// Brief: Mounting Instrument
FUNCTION_BLOCK PUBLIC FB_SlaveCtrlMountInstru EXTENDS FB_SlaveArmCtrlBase
VAR
	// mount status
	m_instruMountStatus :INT := 0;
	m_scopeMountStatus :INT := 0;
	m_ultrasoundMountStatus :INT :=0 ;
	
	// flag if joint is mounted
	m_jointMounted :ARRAY[1..5] OF BOOL := [5(FALSE)];
	
	// instrument mount motion range
	m_mountMotionAng :Vec5d :=[5(pi)];
	
	// instrument mount direction
	m_mountDir :Vec5i :=[1, 1, 1, 1, 1];
	
	// mount motion planning
	m_jntOTG :ARRAY[1..5] OF FB_secOrdTrajFilter;
	m_instruMountVel :LREAL := 4*PI;
	m_instruMountAcc :LREAL := 8*PI;
	
	//Joint 4 half-range angle of instrument
	m_instruJnt4HalfRangeAng :LREAL := 323*g_deg2Rad;
	
	// joint current threshold which indicate panel is buckled with instrument
	m_maxJntCurrent :Vec5d := [150, 150, 150, 180, 180];
	
	// command mount motion
	m_targetMountPos :Vec8d;
	
	// instrument zero position
	m_instruZeroDeviation :Vec5d;
	
	//ultrasound knife Reduce the current rotation Angle  J3
	m_ultraKnifeRotaAngleJ3 :LREAL := 30*g_deg2Rad;
	
	// ultrasound knife rotate angle zero position
	m_ultraKnifeRotAngZeroPos :LREAL := 4.50567;
	
	// joint position error
	m_jntPosErr :Vec5d;
	
	// endoscope motion angle to original position
	m_scopeJnt4CenterMotionAng :LREAL :=175*g_deg2Rad;
	m_scopeJnt5CenterMotionAng :LREAL :=150*g_deg2Rad;
	
	//instrument clamp error Id
	m_instruClampErrId : UINT;
	m_instruClampTime : LREAL;
	m_noCurrentTime : LREAL :=3;
	m_notReturnToZero : LREAL :=5;
END_VAR

// override this function in each exact controller
METHOD PROTECTED calcCmdJntPos : BOOL
VAR_IN_OUT CONSTANT
	i_endoscopePose : ST_Frame;
	i_masterStatus :ST_MasterStatus;
	i_setupStatus: ST_SetupStatus;
	i_slaveArm :FB_SlaveArm;
END_VAR

VAR 
END_VAR
// return directly if instrument/endoscope is not readed
IF i_slaveArm.instrument.onChipData.m_Error OR m_instruClampErrId >0  THEN
	return;
END_IF

IF i_slaveArm.instrument.onChipData.m_InstruReadSucceed AND InstruType_endoscope = i_slaveArm.instrument.m_instruType THEN
	mountEndoscope(i_slaveArm);
ELSIF i_slaveArm.instrument.onChipData.m_InstruReadSucceed AND (InstruType_UltrasoundKnifeS = i_slaveArm.instrument.m_instruType OR InstruType_UltrasoundKnifeU = i_slaveArm.instrument.m_instruType) THEN
	mountUltraKnife(i_slaveArm);
ELSE
	mountInstrument(i_slaveArm);
END_IF
m_instruClampErrId := instruClampStatus(i_slaveArm);
END_METHOD

METHOD PUBLIC init : BOOL
VAR_IN_OUT CONSTANT
	i_slaveArm	:FB_SlaveArm;
END_VAR
VAR_IN_OUT 
	r_slaveArmCtrlCmd :ST_SlaveArmCtrlCmds;
END_VAR

VAR
	i : INT;
END_VAR
// check if to hold the command joint position unchanged
m_holdLastCmds := checkToHoldLastCmds(i_slaveArm);

SUPER^.Init(i_slaveArm,r_slaveArmCtrlCmd);
m_jntOPMode[4] := DriverOPMode_PosTrq;
m_jntOPMode[5] := DriverOPMode_PosTrq;
m_jntOPMode[6] := DriverOPMode_PosTrq;
m_jntOPMode[7] := DriverOPMode_PosTrq;
m_jntOPMode[8] := DriverOPMode_PosTrq;

FOR i:=1 TO 5 DO
	m_targetMountPos[i+3]:=m_cmdJntPos[i+3];
	m_jntOTG[i].init(m_targetMountPos[i+3], 0,m_instruMountVel, m_instruMountAcc, g_slaveArmCtrlCycleTime);
	m_jointMounted[i]:=FALSE;
END_FOR

m_instruMountStatus:=0;
m_scopeMountStatus:=0;
m_ultrasoundMountStatus:=0;
m_instruClampErrId := 0;
m_instruClampTime := 0;
// update commands to arm
copyCmds(r_slaveArmCtrlCmd);
END_METHOD

PROPERTY instruClampErrId :  UINT
GET
instruClampErrId := m_instruClampErrId;
END_GET
END_PROPERTY

METHOD instruClampStatus : UINT
VAR_IN_OUT CONSTANT
	i_slaveArm :FB_SlaveArm;
END_VAR
//m_instruClampErrId=1 instrumen clamp the current does not reach the set value
//m_instruClampErrId=2 instrumen clamp position does not return to zero
m_instruClampTime := LIMIT(0,m_instruClampTime + g_slaveArmCtrlCycleTime,10);
IF i_slaveArm.instrument.onChipData.m_InstruReadSucceed THEN
	IF InstruType_endoscope = i_slaveArm.instrument.m_instruType THEN
		IF (m_scopeMountStatus=0 OR m_scopeMountStatus=1) AND m_instruClampTime>=m_noCurrentTime  THEN
			instruClampStatus := 1;
		ELSIF m_scopeMountStatus=3 AND m_instruClampTime>=m_notReturnToZero  THEN
			instruClampStatus := 2;
		END_IF
		
	ELSIF (InstruType_UltrasoundKnifeS = i_slaveArm.instrument.m_instruType OR InstruType_UltrasoundKnifeU = i_slaveArm.instrument.m_instruType) THEN
		IF (m_ultrasoundMountStatus=0) AND m_instruClampTime>=m_noCurrentTime  THEN
			instruClampStatus := 1;
		ELSIF (m_scopeMountStatus=3) AND m_instruClampTime>=m_notReturnToZero  THEN
			instruClampStatus := 2;
		END_IF
			
	ELSE
		IF (m_instruMountStatus=0) AND m_instruClampTime>=m_noCurrentTime  THEN
			instruClampStatus := 1;
		ELSIF (m_instruMountStatus=3) AND m_instruClampTime>=m_notReturnToZero  THEN
			instruClampStatus := 2;
		END_IF
	END_IF
END_IF
END_METHOD

METHOD mountEndoscope : BOOL
VAR_IN_OUT CONSTANT
	i_slaveArm :FB_SlaveArm;
END_VAR

VAR 
	i :INT;
	curJntPos :Vec8d;
END_VAR
curJntPos := i_slaveArm.curJntPos;

CASE m_scopeMountStatus OF
	//fix scope lock joint(joint 7)
	0:
		// other joints stay still
		FOR i:=1 TO 3 DO
			m_jointMounted[i] := TRUE;
			m_targetMountPos[i+3]:=curJntPos[i+3];
			m_jntOTG[i].init(m_targetMountPos[i+3], 0,m_instruMountVel, m_instruMountAcc, g_slaveArmCtrlCycleTime);
		END_FOR
	
		// check if buckled
		m_jointMounted[4]:=FALSE; 
		m_jointMounted[5]:=FALSE; 
		IF ABS(i_slaveArm.filtJntCurrent[7])> m_maxJntCurrent[4] THEN 
			m_jointMounted[4]:=TRUE;
			m_targetMountPos[7]:=curJntPos[7];
			m_jntOTG[4].init(m_targetMountPos[7], 0,m_instruMountVel, m_instruMountAcc, g_slaveArmCtrlCycleTime);
			m_scopeMountStatus:=1;
		ELSE
			m_targetMountPos[7]:=curJntPos[7]+m_mountMotionAng[4];
		END_IF

	1: // buckle scope rotate joint (joint 8)
		m_jointMounted[5]:=FALSE; 
		IF ABS(i_slaveArm.filtJntCurrent[8])> m_maxJntCurrent[5] THEN 
			m_jointMounted[5]:=TRUE;
			m_targetMountPos[8]:=curJntPos[8];
			m_jntOTG[5].init(m_targetMountPos[8], 0,m_instruMountVel, m_instruMountAcc, g_slaveArmCtrlCycleTime);
			m_scopeMountStatus:=2;
		ELSE
			m_targetMountPos[8]:=curJntPos[8]+m_mountMotionAng[5];
		END_IF
	

	2:// move back to zero position
		m_targetMountPos[7]:= curJntPos[7]-m_scopeJnt4CenterMotionAng;
		m_targetMountPos[8]:= curJntPos[8]-m_scopeJnt5CenterMotionAng;
		m_scopeMountStatus :=3;
		
		
	3:
		IF ABS(m_targetMountPos[7]-curJntPos[7]) <GVL_SlaveControlParameters.g_jntCtrlAngTolHigh AND 
				ABS(m_targetMountPos[8]-curJntPos[8]) <GVL_SlaveControlParameters.g_jntCtrlAngTolHigh THEN
			// record current joint position as offset for instrument
			i_slaveArm.instrument.initInstruJntPos(i_slaveArm.curJntPos);
			m_isFinished := TRUE;
		END_IF
		
END_CASE

// traj plan
FOR i:=1 TO 5 DO
	m_jntOTG[i].run(m_targetMountPos[i+3],0.0, o_cmdAcc=>m_cmdJntAcc[3+i],o_cmdVel=>m_cmdJntVel[3+i],o_cmdPos=>m_cmdJntPos[i+3]);
END_FOR
END_METHOD

METHOD mountInstrument : BOOL
VAR_IN_OUT CONSTANT
	i_slaveArm :FB_SlaveArm;
END_VAR

VAR 
	i :INT;
	curJntPos :Vec8d;
END_VAR
curJntPos := i_slaveArm.curJntPos;

// joint4 stay still if instrument has only on finger
IF i_slaveArm.instrument.m_isSingleFinger THEN
	m_jointMounted[1]:=TRUE;
END_IF

CASE m_instruMountStatus OF
	// To lock panel with instrument
	0:
		//buckle panel with instrument
		FOR i:=1 TO 4 DO
			// check if buckled 
			IF ABS(i_slaveArm.filtJntCurrent[i+3])> m_maxJntCurrent[i] THEN 
				m_jointMounted[i]:=TRUE;
				m_targetMountPos[i+3]:=curJntPos[i+3];
				m_jntOTG[i].init(m_targetMountPos[i+3], 0,m_instruMountVel, m_instruMountAcc, g_slaveArmCtrlCycleTime);
			END_IF
			
			// set target joint position
			IF FALSE = m_jointMounted[i] THEN
				IF i = 4 THEN
					m_targetMountPos[i+3]:=curJntPos[i+3]+m_mountMotionAng[i];
				ELSE
					m_targetMountPos[i+3]:=curJntPos[i+3]-m_mountMotionAng[i];
				END_IF
				
			END_IF
		END_FOR
		
		
		// check transition condition
		IF (m_jointMounted[1] AND m_jointMounted[2] AND m_jointMounted[3] AND m_jointMounted[4])  THEN
			IF i_slaveArm.instrument.onChipData.m_InstruReadSucceed THEN//Check whether the data is read successfully
				m_instruMountStatus:=1;
			END_IF
		END_IF
	
	1:// calculation deviates from the instrument zero position
		FOR i:=1 TO 4 DO
			m_instruZeroDeviation[i] :=  i_slaveArm.linkSingle[i+3] - i_slaveArm.instrument.onChipData.m_InstruPos[i];
		END_FOR
		m_instruMountStatus :=2;
	
	
	2:// move back to zero position
		FOR i:=1 TO 3 DO//J1-3
			IF m_instruZeroDeviation[i]>pi THEN
				m_instruZeroDeviation[i] := m_instruZeroDeviation[i] - 2*PI;
			ELSIF m_instruZeroDeviation[i]<-pi THEN
				m_instruZeroDeviation[i] := m_instruZeroDeviation[i] + 2*PI;
			END_IF
		END_FOR
		
		//joint4
		IF m_instruZeroDeviation[4]>0 AND m_instruZeroDeviation[4] < pi THEN
			m_instruZeroDeviation[4] := m_instruZeroDeviation[4] - 2*pi;
		ELSIF m_instruZeroDeviation[4]<0 AND m_instruZeroDeviation[4] > -pi THEN
			m_instruZeroDeviation[4] := m_instruZeroDeviation[4] + 2*pi;
		END_IF
		
		// set target joint position
		FOR i:=1 TO 4 DO
			m_targetMountPos[i+3]:=curJntPos[i+3] - m_instruZeroDeviation[i];
		END_FOR
		m_instruMountStatus :=3;
	
	3: // make fingers is closed
		//m_instruMountStatus :=4;
		FOR i:=1 TO 4 DO 
			m_jointMounted[i]:=FALSE;
			m_jntPosErr[i]:=m_targetMountPos[i+3]-curJntPos[i+3];
			IF ABS(m_jntPosErr[i]) <GVL_SlaveControlParameters.g_jntCtrlAngTolLow OR 
					ABS( i_slaveArm.linkSingle[i+3] - i_slaveArm.instrument.onChipData.m_InstruPos[i]) <5*g_deg2rad THEN
				m_jointMounted[i]:=TRUE;
				//EXIT;
			END_IF
		END_FOR
		
		IF ABS(i_slaveArm.filtJntCurrent[7])> m_maxJntCurrent[4] AND ABS(i_slaveArm.curJntVel[7])< 1*g_deg2rad AND
				ABS( i_slaveArm.linkSingle[7] - i_slaveArm.instrument.onChipData.m_InstruPos[4]) >10*g_deg2rad AND NOT m_jointMounted[4] THEN 
			m_instruZeroDeviation[4] :=  i_slaveArm.linkSingle[7] - i_slaveArm.instrument.onChipData.m_InstruPos[4];
			m_jointMounted[4]:=TRUE;
			IF m_instruZeroDeviation[4]>=0 AND m_instruZeroDeviation[4] < pi THEN
				m_instruZeroDeviation[4] := m_instruZeroDeviation[4] - 2*pi;
			ELSIF m_instruZeroDeviation[4]<0 AND m_instruZeroDeviation[4] > -pi THEN
				m_instruZeroDeviation[4] := m_instruZeroDeviation[4] + 2*pi;	
			END_IF
		ELSE
			m_instruZeroDeviation[4] := 0;
		END_IF
		
		IF (m_jointMounted[1] AND m_jointMounted[2] AND m_jointMounted[3] AND m_jointMounted[4])  THEN
			m_instruMountStatus :=4;
		END_IF
		
		IF m_instruMountStatus =4 AND NOT( i_slaveArm.instrument.m_isSingleFinger) THEN
			m_targetMountPos[4] := curJntPos[4]+g_gripperCloseAng;
			m_targetMountPos[5] := curJntPos[5]+g_gripperCloseAng;
			m_targetMountPos[7] := curJntPos[7]-m_instruZeroDeviation[4];
		END_IF
		
	4:
		m_isFinished :=  ABS(m_targetMountPos[4]-curJntPos[4]) < GVL_SlaveControlParameters.g_jntCtrlAngTolLow AND
			 ABS(m_targetMountPos[5]-curJntPos[5]) < GVL_SlaveControlParameters.g_jntCtrlAngTolLow AND ABS(m_targetMountPos[7]-curJntPos[7]) < GVL_SlaveControlParameters.g_jntCtrlAngTolLow;
			 
		// record current joint position as offset for instrument
		i_slaveArm.instrument.initInstruJntPos(i_slaveArm.curJntPos);

END_CASE

// traj plan
FOR i:=1 TO 4 DO
	m_jntOTG[i].run(m_targetMountPos[i+3],0.0, o_cmdAcc=>m_cmdJntAcc[3+i],o_cmdVel=>m_cmdJntVel[3+i],o_cmdPos=>m_cmdJntPos[i+3]);
END_FOR
END_METHOD

METHOD mountUltraKnife : BOOL
VAR_IN_OUT CONSTANT
	i_slaveArm :FB_SlaveArm;
END_VAR

VAR 
	i :INT;
	curJntPos :Vec8d;
END_VAR
curJntPos := i_slaveArm.curJntPos;

m_jointMounted[1]:=TRUE;
m_jointMounted[2]:=TRUE;


CASE m_ultrasoundMountStatus OF 
	// To lock panel with instrument
	0:
		//buckle panel with instrument
		FOR i:=3 TO 5 DO
			// check if buckled 
			IF ABS(i_slaveArm.filtJntCurrent[i+3])> m_maxJntCurrent[i] THEN 
				m_jointMounted[i]:=TRUE;
				m_targetMountPos[i+3]:=curJntPos[i+3];
				m_jntOTG[i].init(m_targetMountPos[i+3], 0,m_instruMountVel, m_instruMountAcc, g_slaveArmCtrlCycleTime);
			END_IF
			
			// set target joint position
			IF FALSE = m_jointMounted[i] THEN
				IF i = 5 THEN
					m_targetMountPos[i+3]:=curJntPos[i+3]+m_mountMotionAng[i];
				ELSE
					m_targetMountPos[i+3]:=curJntPos[i+3]-m_mountMotionAng[i];
				END_IF
				
			END_IF
		END_FOR

		// check transition condition
		IF ( m_jointMounted[3] AND m_jointMounted[4] AND m_jointMounted[5] )  THEN
			IF i_slaveArm.instrument.onChipData.m_InstruReadSucceed THEN//Check whether the data is read successfully
				m_ultrasoundMountStatus:=1;
			END_IF
		END_IF

	1:
		//m_jntOPMode[8] := DriverOPMode_Trq;
		// calculation deviates from the instrument zero position
		m_instruZeroDeviation[3] :=  m_ultraKnifeRotaAngleJ3;
		m_instruZeroDeviation[4] :=  i_slaveArm.linkSingle[7] - m_ultraKnifeRotAngZeroPos;
		m_ultrasoundMountStatus :=2;
		
	2:// move back to zero position
		//joint4
		IF m_instruZeroDeviation[4]>0 AND m_instruZeroDeviation[4] < pi THEN
			m_instruZeroDeviation[4] := m_instruZeroDeviation[4] - 2*pi;
		ELSIF m_instruZeroDeviation[4]<0 AND m_instruZeroDeviation[4] > -pi THEN
			m_instruZeroDeviation[4] := m_instruZeroDeviation[4] + 2*pi;
		END_IF
	
		// set target joint position
		m_targetMountPos[6]:=curJntPos[6] + m_instruZeroDeviation[3];
		m_targetMountPos[7]:=curJntPos[7] - m_instruZeroDeviation[4];
		m_targetMountPos[8]:=curJntPos[8] - m_instruZeroDeviation[4];

		m_ultrasoundMountStatus :=3;

	3:
		// joint8 in passive mode
		m_jntOPMode[8] := DriverOPMode_Trq;
		
		m_isFinished:=TRUE;
		FOR i:=3 TO 4 DO 
			m_jntPosErr[i]:=m_targetMountPos[i+3]-curJntPos[i+3];
			IF ABS(m_jntPosErr[i]) >GVL_SlaveControlParameters.g_jntCtrlAngTolLow  THEN
				m_isFinished := FALSE;
				EXIT;
			END_IF
		END_FOR	
		
		// record current joint position as offset for instrument
		i_slaveArm.instrument.initInstruJntPos(i_slaveArm.curJntPos);

END_CASE


// traj plan
FOR i:=1 TO 5 DO
	m_jntOTG[i].run(m_targetMountPos[i+3],0.0, o_cmdAcc=>m_cmdJntAcc[3+i],o_cmdVel=>m_cmdJntVel[3+i],o_cmdPos=>m_cmdJntPos[i+3]);
END_FOR
END_METHOD

END_FUNCTION_BLOCK

(* stored: Version 1.1.0.1, ProductVersion 3.1.4024.11
   POU FB_SlaveCtrlMountInstru: Id {db93de24-03af-45f5-8edb-e02a943fe1f8}, SpecialFunc None
   Method calcCmdJntPos: Id {106b8ce6-26fa-4bca-bfc9-20f8cdf00f0e}
   Method init: Id {85ccbdcb-d27d-4162-a6ec-e8e93d30dbc6}
   Property instruClampErrId: Id {f1028432-c4d8-4b7e-a34b-a7a30fe5b17a}
   Get Get: Id {4e5cc1ce-1710-4380-ad0f-4115ae9409f8}
   Method instruClampStatus: Id {59da6779-a8b0-41c0-b6ac-feaa3bdf40f7}
   Method mountEndoscope: Id {924322f0-f77b-4627-9090-85580b93061c}
   Method mountInstrument: Id {cbdcc411-d3ae-4c70-8c1a-fbdc24e77583}
   Method mountUltraKnife: Id {6b01324c-5b90-4e88-a0ef-19a2c0251538} *)
